Fanuc KAREL source: kd00061.KL

-- PROVISIONAL review KL for V770-1; original PC SHA256 b8f8d7b8b98e55a4358c2076d73c79b052936b3f555f3da6dc2347c9ccaee028
-- Incomplete behavior may be omitted. Consult companion uncertainty JSON. Do not deploy.
PROGRAM KD00061
%NOLOCKGROUP
VAR
  I : INTEGER
  J : INTEGER
  B : BOOLEAN
  R : REAL
  S : STRING[80]
BEGIN
  -- UNRESOLVED_PC offsets 5-18; opcodes 9D,81,18,9D,1B,9D,12,9D,13,04
  -- UNRESOLVED_PC offsets 23-27; opcodes 7F
END KD00061
